ABB RAPID module: lab01_main.mod

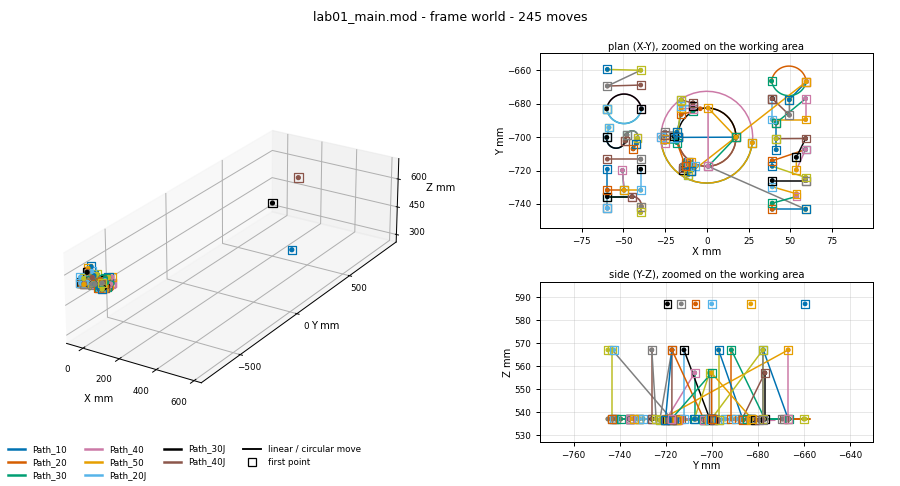
[picture p0: tool path of lab01_main.mod in frame world, 245 of 245 moves have a stored position in this frame; points joined in program order, loops and branches not executed]
MODULE Module1
    CONST robtarget Target_20J:=[[134.579,32.471,0],[1,0,0,0],[0,0,0,0],[9E+09,9E+09,9E+09,9E+09,9E+09,9E+09]];
    CONST robtarget Target_30J:=[[134.579,39.359,0],[1,0,0,0],[0,0,0,0],[9E+09,9E+09,9E+09,9E+09,9E+09,9E+09]];
    CONST robtarget Target_40J:=[[134.579,39.359,0],[1,0,0,0],[0,0,0,0],[9E+09,9E+09,9E+09,9E+09,9E+09,9E+09]];
    CONST robtarget Target_50J:=[[119.781,39.359,0],[1,0,0,0],[0,0,0,0],[9E+09,9E+09,9E+09,9E+09,9E+09,9E+09]];
    CONST robtarget Target_10H:=[[-531.42717004,745,-69.059806194],[0.965925826,0,-0.258819045,0],[0,0,0,0],[9E+09,9E+09,9E+09,9E+09,9E+09,9E+09]];
    CONST robtarget Target_60J:=[[115.729,37.754,0],[1,0,0,0],[0,0,0,0],[9E+09,9E+09,9E+09,9E+09,9E+09,9E+09]];
    CONST robtarget Target_70J:=[[114.303,33.443,0],[1,0,0,0],[0,0,0,0],[9E+09,9E+09,9E+09,9E+09,9E+09,9E+09]];
    CONST robtarget Target_80J:=[[114.692,29.91,0],[1,0,0,0],[0,0,0,0],[9E+09,9E+09,9E+09,9E+09,9E+09,9E+09]];
    CONST robtarget Target_10:=[[606.42717004,0,579.059806194],[0.258819045,0,0.965925826,0],[0,0,0,0],[9E+09,9E+09,9E+09,9E+09,9E+09,9E+09]];
    CONST robtarget Target_30:=[[134.579,39.359,0],[0.707106781,0,0,0.707106781],[0,0,0,0],[9E+09,9E+09,9E+09,9E+09,9E+09,9E+09]];
    CONST robtarget Target_20:=[[134.579,32.471,0],[0.707106781,0,0,0.707106781],[0,0,0,0],[9E+09,9E+09,9E+09,9E+09,9E+09,9E+09]];
    CONST robtarget Target_40:=[[119.781,39.359,0],[0.707106781,0,0,0.707106781],[0,0,0,0],[9E+09,9E+09,9E+09,9E+09,9E+09,9E+09]];
    CONST robtarget Target_50:=[[115.729,37.754,0],[0.707106781,0,0,0.707106781],[0,0,0,0],[9E+09,9E+09,9E+09,9E+09,9E+09,9E+09]];
    CONST robtarget Target_60:=[[114.303,33.443,0],[0.707106781,0,0,0.707106781],[0,0,0,0],[9E+09,9E+09,9E+09,9E+09,9E+09,9E+09]];
    CONST robtarget Target_70:=[[114.692,29.91,0],[0.707106781,0,0,0.707106781],[0,0,0,0],[9E+09,9E+09,9E+09,9E+09,9E+09,9E+09]];
    CONST robtarget Target_80:=[[114.692,29.91,-30],[0.707106781,0,0,0.707106781],[0,0,0,0],[9E+09,9E+09,9E+09,9E+09,9E+09,9E+09]];
    CONST robtarget Target_90:=[[134.579,55.793,0],[0.707106781,0,0,0.707106781],[0,0,0,0],[9E+09,9E+09,9E+09,9E+09,9E+09,9E+09]];
    CONST robtarget Target_100:=[[134.579,43.281,0],[0.707106781,0,0,0.707106781],[0,0,0,0],[9E+09,9E+09,9E+09,9E+09,9E+09,9E+09]];
    CONST robtarget Target_110:=[[124.579,43.281,0],[0.707106781,0,0,0.707106781],[0,0,0,0],[9E+09,9E+09,9E+09,9E+09,9E+09,9E+09]];
    CONST robtarget Target_120:=[[125.551,55.129,0],[0.707106781,0,0,0.707106781],[0,0,0,0],[9E+09,9E+09,9E+09,9E+09,9E+09,9E+09]];
    CONST robtarget Target_130:=[[114.579,43.281,0],[0.707106781,0,0,0.707106781],[0,0,0,0],[9E+09,9E+09,9E+09,9E+09,9E+09,9E+09]];
    CONST robtarget Target_140:=[[114.579,55.793,0],[0.707106781,0,0,0.707106781],[0,0,0,0],[9E+09,9E+09,9E+09,9E+09,9E+09,9E+09]];
    CONST robtarget Target_160:=[[114.579,55.793,-50],[0.707106781,0,0,0.707106781],[0,0,0,0],[9E+09,9E+09,9E+09,9E+09,9E+09,9E+09]];
    CONST robtarget Target_170:=[[134.579,61.806,0],[0.707106781,0,0,0.707106781],[0,0,0,0],[9E+09,9E+09,9E+09,9E+09,9E+09,9E+09]];
    CONST robtarget Target_180:=[[114.579,61.806,0],[0.707106781,0,0,0.707106781],[0,0,0,0],[9E+09,9E+09,9E+09,9E+09,9E+09,9E+09]];
    CONST robtarget Target_190:=[[114.579,61.806,-50],[0.707106781,0,0,0.707106781],[0,0,0,0],[9E+09,9E+09,9E+09,9E+09,9E+09,9E+09]];
    CONST robtarget Target_200:=[[133.639,80.801,0],[0.707106781,0,0,0.707106781],[0,0,0,0],[9E+09,9E+09,9E+09,9E+09,9E+09,9E+09]];
    CONST robtarget Target_210:=[[134.935,74.853,0],[0.707106781,0,0,0.707106781],[0,0,0,0],[9E+09,9E+09,9E+09,9E+09,9E+09,9E+09]];
    CONST robtarget Target_220:=[[133.29,70.023,0],[0.707106781,0,0,0.707106781],[0,0,0,0],[9E+09,9E+09,9E+09,9E+09,9E+09,9E+09]];
    CONST robtarget Target_230:=[[123.833,72.73,0],[0.707106781,0,0,0.707106781],[0,0,0,0],[9E+09,9E+09,9E+09,9E+09,9E+09,9E+09]];
    CONST robtarget Target_240:=[[122.925,76.344,0],[0.707106781,0,0,0.707106781],[0,0,0,0],[9E+09,9E+09,9E+09,9E+09,9E+09,9E+09]];
    CONST robtarget Target_250:=[[119.862,78.808,0],[0.707106781,0,0,0.707106781],[0,0,0,0],[9E+09,9E+09,9E+09,9E+09,9E+09,9E+09]];
    CONST robtarget Target_260:=[[116.524,74.351,0],[0.707106781,0,0,0.707106781],[0,0,0,0],[9E+09,9E+09,9E+09,9E+09,9E+09,9E+09]];
    CONST robtarget Target_270:=[[117.204,71.15,0],[0.707106781,0,0,0.707106781],[0,0,0,0],[9E+09,9E+09,9E+09,9E+09,9E+09,9E+09]];
    CONST robtarget Target_280:=[[119.117,68.078,0],[0.707106781,0,0,0.707106781],[0,0,0,0],[9E+09,9E+09,9E+09,9E+09,9E+09,9E+09]];
    CONST robtarget Target_290:=[[119.117,67.981,-50],[0.707106781,0,0,0.707106781],[0,0,0,0],[9E+09,9E+09,9E+09,9E+09,9E+09,9E+09]];
    CONST robtarget Target_300:=[[135,91.984,0],[0.707106781,0,0,0.707106781],[0,0,0,0],[9E+09,9E+09,9E+09,9E+09,9E+09,9E+09]];
    CONST robtarget Target_310:=[[124.579,83.151,0],[0.707106781,0,0,0.707106781],[0,0,0,0],[9E+09,9E+09,9E+09,9E+09,9E+09,9E+09]];
    CONST robtarget Target_320:=[[114.157,91.984,0],[0.707106781,0,0,0.707106781],[0,0,0,0],[9E+09,9E+09,9E+09,9E+09,9E+09,9E+09]];
    CONST robtarget Target_330:=[[124.579,100.834,0],[0.707106781,0,0,0.707106781],[0,0,0,0],[9E+09,9E+09,9E+09,9E+09,9E+09,9E+09]];
    CONST robtarget Target_340:=[[135,91.984,-50],[0.707106781,0,0,0.707106781],[0,0,0,0],[9E+09,9E+09,9E+09,9E+09,9E+09,9E+09]];
    CONST robtarget Target_360:=[[114.579,106.231,0],[0.707106781,0,0,0.707106781],[0,0,0,0],[9E+09,9E+09,9E+09,9E+09,9E+09,9E+09]];
    CONST robtarget Target_350:=[[134.579,105.639,0],[0.707106781,0,0,0.707106781],[0,0,0,0],[9E+09,9E+09,9E+09,9E+09,9E+09,9E+09]];
    CONST robtarget Target_370:=[[114.579,115.08,0],[0.707106781,0,0,0.707106781],[0,0,0,0],[9E+09,9E+09,9E+09,9E+09,9E+09,9E+09]];
    CONST robtarget Target_380:=[[134.579,115.582,0],[0.707106781,0,0,0.707106781],[0,0,0,0],[9E+09,9E+09,9E+09,9E+09,9E+09,9E+09]];
    CONST robtarget Target_390:=[[134.579,115.582,-50],[0.707106781,0,0,0.707106781],[0,0,0,0],[9E+09,9E+09,9E+09,9E+09,9E+09,9E+09]];
    CONST robtarget Target_400:=[[102.5,75,0],[0.707106781,0,0,0.707106781],[0,0,0,0],[9E+09,9E+09,9E+09,9E+09,9E+09,9E+09]];
    CONST robtarget Target_410:=[[77.953,102.341,0.5],[0.707106781,0,0,0.707106781],[0,0,0,0],[9E+09,9E+09,9E+09,9E+09,9E+09,9E+09]];
    CONST robtarget Target_420:=[[47.704,71.659,0.5],[0.707106781,0,0,0.707106781],[0,0,0,0],[9E+09,9E+09,9E+09,9E+09,9E+09,9E+09]];
    CONST robtarget Target_430:=[[73.18,47.56,0],[0.707106781,0,0,0.707106781],[0,0,0,0],[9E+09,9E+09,9E+09,9E+09,9E+09,9E+09]];
    CONST robtarget Target_440:=[[92.5,75,0],[0.707106781,0,0,0.707106781],[0,0,0,0],[9E+09,9E+09,9E+09,9E+09,9E+09,9E+09]];
    CONST robtarget Target_450:=[[57.5,75,0],[0.707106781,0,0,0.707106781],[0,0,0,0],[9E+09,9E+09,9E+09,9E+09,9E+09,9E+09]];
    CONST robtarget Target_460:=[[78.949,92.049,0],[0.707106781,0,0,0.707106781],[0,0,0,0],[9E+09,9E+09,9E+09,9E+09,9E+09,9E+09]];
    CONST robtarget Target_480:=[[102.5,75,-50],[0.707106781,0,0,0.707106781],[0,0,0,0],[9E+09,9E+09,9E+09,9E+09,9E+09,9E+09]];
    CONST robtarget Target_490:=[[74.168,57.52,0],[0.707106781,0,0,0.707106781],[0,0,0,0],[9E+09,9E+09,9E+09,9E+09,9E+09,9E+09]];
    CONST robtarget Target_500:=[[15.79,31.822,-30],[0.707106781,0,0,0.707106781],[0,0,0,0],[9E+09,9E+09,9E+09,9E+09,9E+09,9E+09]];
    CONST robtarget Target_510:=[[15.79,31.822,0],[0.707106781,0,0,0.707106781],[0,0,0,0],[9E+09,9E+09,9E+09,9E+09,9E+09,9E+09]];
    CONST robtarget Target_520:=[[35.79,31.822,0],[0.707106781,0,0,0.707106781],[0,0,0,0],[9E+09,9E+09,9E+09,9E+09,9E+09,9E+09]];
    CONST robtarget Target_530:=[[35.79,35.453,0],[0.707106781,0,0,0.707106781],[0,0,0,0],[9E+09,9E+09,9E+09,9E+09,9E+09,9E+09]];
    CONST robtarget Target_540:=[[21.301,39.472,0],[0.707106781,0,0,0.707106781],[0,0,0,0],[9E+09,9E+09,9E+09,9E+09,9E+09,9E+09]];
    CONST robtarget Target_550:=[[21.301,41.093,0],[0.707106781,0,0,0.707106781],[0,0,0,0],[9E+09,9E+09,9E+09,9E+09,9E+09,9E+09]];
    CONST robtarget Target_560:=[[35.79,45.274,0],[0.707106781,0,0,0.707106781],[0,0,0,0],[9E+09,9E+09,9E+09,9E+09,9E+09,9E+09]];
    CONST robtarget Target_570:=[[35.79,48.97,0],[0.707106781,0,0,0.707106781],[0,0,0,0],[9E+09,9E+09,9E+09,9E+09,9E+09,9E+09]];
    CONST robtarget Target_580:=[[15.79,48.97,0],[0.707106781,0,0,0.707106781],[0,0,0,0],[9E+09,9E+09,9E+09,9E+09,9E+09,9E+09]];
    CONST robtarget Target_590:=[[15.79,48.97,-30],[0.707106781,0,0,0.707106781],[0,0,0,0],[9E+09,9E+09,9E+09,9E+09,9E+09,9E+09]];
    CONST robtarget Target_600:=[[15.79,50.866,0],[0.707106781,0,0,0.707106781],[0,0,0,0],[9E+09,9E+09,9E+09,9E+09,9E+09,9E+09]];
    CONST robtarget Target_610:=[[35.79,57.608,0],[0.707106781,0,0,0.707106781],[0,0,0,0],[9E+09,9E+09,9E+09,9E+09,9E+09,9E+09]];
    CONST robtarget Target_620:=[[35.79,60.882,0],[0.707106781,0,0,0.707106781],[0,0,0,0],[9E+09,9E+09,9E+09,9E+09,9E+09,9E+09]];
    CONST robtarget Target_630:=[[15.79,67.625,0],[0.707106781,0,0,0.707106781],[0,0,0,0],[9E+09,9E+09,9E+09,9E+09,9E+09,9E+09]];
    CONST robtarget Target_640:=[[15.79,67.625,-20],[0.707106781,0,0,0.707106781],[0,0,0,0],[9E+09,9E+09,9E+09,9E+09,9E+09,9E+09]];
    CONST robtarget Target_650:=[[21.361,55.365,0],[0.707106781,0,0,0.707106781],[0,0,0,0],[9E+09,9E+09,9E+09,9E+09,9E+09,9E+09]];
    CONST robtarget Target_660:=[[21.382,62.997,0],[0.707106781,0,0,0.707106781],[0,0,0,0],[9E+09,9E+09,9E+09,9E+09,9E+09,9E+09]];
    CONST robtarget Target_670:=[[21.382,62.943,-30],[0.707106781,0,0,0.707106781],[0,0,0,0],[9E+09,9E+09,9E+09,9E+09,9E+09,9E+09]];
    CONST robtarget Target_680:=[[15.79,74.189,0],[0.707106781,0,0,0.707106781],[0,0,0,0],[9E+09,9E+09,9E+09,9E+09,9E+09,9E+09]];
    CONST robtarget Target_690:=[[33.424,74.097,0],[0.707106781,0,0,0.707106781],[0,0,0,0],[9E+09,9E+09,9E+09,9E+09,9E+09,9E+09]];
    CONST robtarget Target_700:=[[33.424,74.055,-20],[0.707106781,0,0,0.707106781],[0,0,0,0],[9E+09,9E+09,9E+09,9E+09,9E+09,9E+09]];
    CONST robtarget Target_710:=[[33.424,67.479,0],[0.707106781,0,0,0.707106781],[0,0,0,0],[9E+09,9E+09,9E+09,9E+09,9E+09,9E+09]];
    CONST robtarget Target_720:=[[33.424,83.556,0],[0.707106781,0,0,0.707106781],[0,0,0,0],[9E+09,9E+09,9E+09,9E+09,9E+09,9E+09]];
    CONST robtarget Target_730:=[[33.424,83.556,-30],[0.707106781,0,0,0.707106781],[0,0,0,0],[9E+09,9E+09,9E+09,9E+09,9E+09,9E+09]];
    CONST robtarget Target_740:=[[15.79,98.095,0],[0.707106781,0,0,0.707106781],[0,0,0,0],[9E+09,9E+09,9E+09,9E+09,9E+09,9E+09]];
    CONST robtarget Target_750:=[[15.79,85.582,0],[0.707106781,0,0,0.707106781],[0,0,0,0],[9E+09,9E+09,9E+09,9E+09,9E+09,9E+09]];
    CONST robtarget Target_760:=[[35.79,85.582,0],[0.707106781,0,0,0.707106781],[0,0,0,0],[9E+09,9E+09,9E+09,9E+09,9E+09,9E+09]];
    CONST robtarget Target_770:=[[35.79,98.095,0],[0.707106781,0,0,0.707106781],[0,0,0,0],[9E+09,9E+09,9E+09,9E+09,9E+09,9E+09]];
    CONST robtarget Target_780:=[[35.79,98.095,-20],[0.707106781,0,0,0.707106781],[0,0,0,0],[9E+09,9E+09,9E+09,9E+09,9E+09,9E+09]];
    CONST robtarget Target_790:=[[25.531,88.24,0],[0.707106781,0,0,0.707106781],[0,0,0,0],[9E+09,9E+09,9E+09,9E+09,9E+09,9E+09]];
    CONST robtarget Target_800:=[[25.579,97.43,0],[0.707106781,0,0,0.707106781],[0,0,0,0],[9E+09,9E+09,9E+09,9E+09,9E+09,9E+09]];
    CONST robtarget Target_810:=[[25.579,97.43,-30],[0.707106781,0,0,0.707106781],[0,0,0,0],[9E+09,9E+09,9E+09,9E+09,9E+09,9E+09]];
    CONST robtarget Target_820:=[[15.378,108.24,0],[0.707106781,0,0,0.707106781],[0,0,0,0],[9E+09,9E+09,9E+09,9E+09,9E+09,9E+09]];
    CONST robtarget Target_830:=[[24.545794471,117.51743745,0],[0.707106781,0,0,0.707106781],[0,0,0,0],[9E+09,9E+09,9E+09,9E+09,9E+09,9E+09]];
    CONST robtarget Target_840:=[[36.211188313,108.651374241,0],[0.707106781,0,0,0.707106781],[0,0,0,0],[9E+09,9E+09,9E+09,9E+09,9E+09,9E+09]];
    CONST robtarget Target_850:=[[25.417582154,99.88143745,0],[0.707106781,0,0,0.707106781],[0,0,0,0],[9E+09,9E+09,9E+09,9E+09,9E+09,9E+09]];
    CONST robtarget Target_860:=[[15.378,108.24,-30],[0.707106781,0,0,0.707106781],[0,0,0,0],[9E+09,9E+09,9E+09,9E+09,9E+09,9E+09]];
    CONST robtarget Target_870:=[[86.451,52.441,0.5],[0.707106781,0,0,0.707106781],[0,0,0,0],[9E+09,9E+09,9E+09,9E+09,9E+09,9E+09]];
    CONST robtarget Target_890:=[[89.117,56.754,0.5],[0.707106781,0,0,0.707106781],[0,0,0,0],[9E+09,9E+09,9E+09,9E+09,9E+09,9E+09]];
    CONST robtarget Target_880:=[[89.302,55.354,0.5],[0.707106781,0,0,0.707106781],[0,0,0,0],[9E+09,9E+09,9E+09,9E+09,9E+09,9E+09]];
    CONST robtarget Target_900:=[[88.422,57.436,0.5],[0.707106781,0,0,0.707106781],[0,0,0,0],[9E+09,9E+09,9E+09,9E+09,9E+09,9E+09]];
    CONST robtarget Target_910:=[[87.783,57.66,0.546],[0.707106781,0,0,0.707106781],[0,0,0,0],[9E+09,9E+09,9E+09,9E+09,9E+09,9E+09]];
    CONST robtarget Target_920:=[[87.728,58.612,0.5],[0.707106781,0,0,0.707106781],[0,0,0,0],[9E+09,9E+09,9E+09,9E+09,9E+09,9E+09]];
    CONST robtarget Target_930:=[[87.299,59.362,0.5],[0.707106781,0,0,0.707106781],[0,0,0,0],[9E+09,9E+09,9E+09,9E+09,9E+09,9E+09]];
    CONST robtarget Target_940:=[[86.474,59.997,0.5],[0.707106781,0,0,0.707106781],[0,0,0,0],[9E+09,9E+09,9E+09,9E+09,9E+09,9E+09]];
    CONST robtarget Target_950:=[[85.487,60.183,0.5],[0.707106781,0,0,0.707106781],[0,0,0,0],[9E+09,9E+09,9E+09,9E+09,9E+09,9E+09]];
    CONST robtarget Target_960:=[[84.601,59.985,0.5],[0.707106781,0,0,0.707106781],[0,0,0,0],[9E+09,9E+09,9E+09,9E+09,9E+09,9E+09]];
    CONST robtarget Target_970:=[[81.843,57.842,0.5],[0.707106781,0,0,0.707106781],[0,0,0,0],[9E+09,9E+09,9E+09,9E+09,9E+09,9E+09]];
    CONST robtarget Target_980:=[[84.366,54.885,0.5],[0.707106781,0,0,0.707106781],[0,0,0,0],[9E+09,9E+09,9E+09,9E+09,9E+09,9E+09]];
    CONST robtarget Target_990:=[[87.79,57.696,0.5],[0.707106781,0,0,0.707106781],[0,0,0,0],[9E+09,9E+09,9E+09,9E+09,9E+09,9E+09]];
    CONST robtarget Target_1020:=[[87.797,57.739,-30],[0.707106781,0,0,0.707106781],[0,0,0,0],[9E+09,9E+09,9E+09,9E+09,9E+09,9E+09]];
    CONST robtarget Target_1010:=[[86.451,52.441,0.5],[0.707106781,0,0,0.707106781],[0,0,0,0],[9E+09,9E+09,9E+09,9E+09,9E+09,9E+09]];
    CONST robtarget Target_1030:=[[92.924,71.772,0.5],[0.707106781,0,0,0.707106781],[0,0,0,0],[9E+09,9E+09,9E+09,9E+09,9E+09,9E+09]];
    CONST robtarget Target_1040:=[[100.024,71.772,0.5],[0.707106781,0,0,0.707106781],[0,0,0,0],[9E+09,9E+09,9E+09,9E+09,9E+09,9E+09]];
    CONST robtarget Target_1050:=[[100.024,73.703,0.5],[0.707106781,0,0,0.707106781],[0,0,0,0],[9E+09,9E+09,9E+09,9E+09,9E+09,9E+09]];
    CONST robtarget Target_1060:=[[94.605,74.279,0.5],[0.707106781,0,0,0.707106781],[0,0,0,0],[9E+09,9E+09,9E+09,9E+09,9E+09,9E+09]];
    CONST robtarget Target_1070:=[[94.605,75.424,0.5],[0.707106781,0,0,0.707106781],[0,0,0,0],[9E+09,9E+09,9E+09,9E+09,9E+09,9E+09]];
    CONST robtarget Target_1080:=[[100.024,76.047,0.5],[0.707106781,0,0,0.707106781],[0,0,0,0],[9E+09,9E+09,9E+09,9E+09,9E+09,9E+09]];
    CONST robtarget Target_1090:=[[100.024,78.002,0.5],[0.707106781,0,0,0.707106781],[0,0,0,0],[9E+09,9E+09,9E+09,9E+09,9E+09,9E+09]];
    CONST robtarget Target_1100:=[[92.924,78.002,0.5],[0.707106781,0,0,0.707106781],[0,0,0,0],[9E+09,9E+09,9E+09,9E+09,9E+09,9E+09]];
    CONST robtarget Target_1110:=[[92.924,78.002,-30],[0.707106781,0,0,0.707106781],[0,0,0,0],[9E+09,9E+09,9E+09,9E+09,9E+09,9E+09]];
    CONST robtarget Target_1120:=[[90.373,88.629,0.5],[0.707106781,0,0,0.707106781],[0,0,0,0],[9E+09,9E+09,9E+09,9E+09,9E+09,9E+09]];
    CONST robtarget Target_1130:=[[83.273,90.441,0],[0.707106781,0,0,0.707106781],[0,0,0,0],[9E+09,9E+09,9E+09,9E+09,9E+09,9E+09]];
    CONST robtarget Target_1140:=[[83.273,92.124,0.5],[0.707106781,0,0,0.707106781],[0,0,0,0],[9E+09,9E+09,9E+09,9E+09,9E+09,9E+09]];
    CONST robtarget Target_1150:=[[90.373,92.156,0.5],[0.707106781,0,0,0.707106781],[0,0,0,0],[9E+09,9E+09,9E+09,9E+09,9E+09,9E+09]];
    CONST robtarget Target_1160:=[[90.373,93.77,0.5],[0.707106781,0,0,0.707106781],[0,0,0,0],[9E+09,9E+09,9E+09,9E+09,9E+09,9E+09]];
    CONST robtarget Target_1170:=[[83.273,93.784,0.5],[0.707106781,0,0,0.707106781],[0,0,0,0],[9E+09,9E+09,9E+09,9E+09,9E+09,9E+09]];
    CONST robtarget Target_1180:=[[83.273,95.476,0.5],[0.707106781,0,0,0.707106781],[0,0,0,0],[9E+09,9E+09,9E+09,9E+09,9E+09,9E+09]];
    CONST robtarget Target_1190:=[[90.367,97.258,0.5],[0.707106781,0,0,0.707106781],[0,0,0,0],[9E+09,9E+09,9E+09,9E+09,9E+09,9E+09]];
    CONST robtarget Target_1200:=[[90.307,97.243,-30],[0.707106781,0,0,0.707106781],[0,0,0,0],[9E+09,9E+09,9E+09,9E+09,9E+09,9E+09]];
    CONST robtarget Target_1210:=[[92.5,74.875,0],[0.707106781,0,0,0.707106781],[0,0,0,0],[9E+09,9E+09,9E+09,9E+09,9E+09,9E+09]];
    CONST robtarget Target_1220:=[[57.5,75.002,0],[0.707106781,0,0,0.707106781],[0,0,0,0],[9E+09,9E+09,9E+09,9E+09,9E+09,9E+09]];
    CONST robtarget Target_1230:=[[57.5,74.962,-20],[0.707106781,0,0,0.707106781],[0,0,0,0],[9E+09,9E+09,9E+09,9E+09,9E+09,9E+09]];
    CONST robtarget Target_1240:=[[74.192,57.519,0],[0.707106781,0,0,0.707106781],[0,0,0,0],[9E+09,9E+09,9E+09,9E+09,9E+09,9E+09]];
    CONST robtarget Target_1250:=[[74.241,92.484,0],[0.707106781,0,0,0.707106781],[0,0,0,0],[9E+09,9E+09,9E+09,9E+09,9E+09,9E+09]];
    PERS tooldata Tool_JM:=[TRUE,[[36.916,0,136.94],[0.965925826,0,0.258819045,0]],[0.1,[0,0,1],[1,0,0,0],0,0,0]];
    TASK PERS wobjdata Workobject_4:=[FALSE,TRUE,"",[[0,-100,27],[1,0,0,0]],[[75,-675,510],[0,0,1,0]]];
    CONST robtarget Target_1260:=[[134.579,32.471,-30],[0.707106781,0,0,0.707106781],[0,0,0,0],[9E+09,9E+09,9E+09,9E+09,9E+09,9E+09]];
    CONST robtarget Target_1270:=[[74.522025646,1604.781854023,155.867635961],[0.664355676,-0.23027169,-0.237213164,-0.670325592],[1,0,-1,0],[9E+09,9E+09,9E+09,9E+09,9E+09,9E+09]];
    CONST robtarget Target_1280:=[[-35.006958294,1674.86910456,16.96090151],[0.661721738,-0.310193659,-0.350423362,-0.585753961],[0,0,-1,1],[9E+09,9E+09,9E+09,9E+09,9E+09,9E+09]];

    PROC main()

        WHILE TRUE DO

            IF DI_01 = 1 THEN
                Set DO_01;
                WaitTime(4.9);
                Reset DO_01;
                Path_10;
                Path_1110;
                Path_20J;
                Path_30J;
                Path_40J;
                Path_50J;
                Path_60;
                Path_70E;
                Path_80E;
                Path_90E;
                Path_100E;
                Path_110E;
                Path_120E;
                Path_120;
                Path_130I;
                Path_140;
                Path_150S;
                Path_160S;
                Path_170S;
                Path_180S;
                Path_190S;
                Path_200S;
                Path_210;
                Path_220O;
                Path_230O;
                Path_240;
                Path_250N;
                Path_260N;
                Path_270N;
                Path_280;
                Path_290L;
                Path_300;
                Path_310;
                Path_320;
                Path_330;
                Path_340;
                Path_350;
                Path_360;
                Path_370;
                Path_380;
                Path_390;
                Path_400;
                Path_410;
                Path_420;
                Path_430;
                Path_440;
                Path_450;
                Path_460;
                Path_470;
                Path_480;
                Path_490;
                Path_500;
                Path_510;
                Path_520;
                Path_530;
                Path_540;
                Path_550;
                Path_560;
                Path_570;
                Path_580;
                Path_590;
                Path_600;
                Path_610;
                Path_620;
                Path_630;
                Path_640;
                Path_650;
                Path_660;
                Path_670;
                Path_680;
                Path_690;
                Path_700;
                Path_710;
                Path_720;
                Path_730;
                Path_740;
                Path_750;
                Path_760;
                Path_770;
                Path_780;
                Path_790;
                Path_800;
                Path_810;
                Path_820;
                Path_830;
                Path_840;
                Path_850;
                Path_860;
                Path_870;
                Path_880;
                Path_890;
                Path_900;
                Path_910;
                Path_920;
                Path_930;
                Path_940;
                Path_950;
                Path_960;
                Path_970;
                Path_980;
                Path_990;
                Path_1000;
                Path_1010;
                Path_1020;
                Path_1030;
                Path_1040;
                Path_1050;
                Path_1060;
                Path_1070;
                Path_1080;
                Path_1090;
                Path_1100;


                Path_10;

                Reset DO_01;


            ENDIF

            IF DI_02 = 1 THEN
                Set DO_02;
                Path_1130;
                Reset DO_02;

            ENDIF




        ENDWHILE

    ENDPROC
    PROC Path_10()
        MoveJ Target_10,v100,z10,Tool_JM\WObj:=wobj0;
    ENDPROC
    PROC Path_20()
        MoveL Target_20,v100,z10,Tool_JM\WObj:=Workobject_4;
        MoveL Target_30,v100,z10,Tool_JM\WObj:=Workobject_4;
    ENDPROC
    PROC Path_30()
        MoveL Target_30,v100,z10,Tool_JM\WObj:=Workobject_4;
        MoveL Target_40,v100,z10,Tool_JM\WObj:=Workobject_4;
    ENDPROC
    PROC Path_40()
        MoveJ Target_40,v100,z10,Tool_JM\WObj:=Workobject_4;
        MoveC Target_50,Target_60,v100,z10,Tool_JM\WObj:=Workobject_4;
    ENDPROC
    PROC Path_50()
        MoveL Target_60,v100,z10,Tool_JM\WObj:=Workobject_4;
        MoveL Target_70,v100,z10,Tool_JM\WObj:=Workobject_4;
    ENDPROC
    PROC Path_20J()
        MoveL Target_20,v100,z10,Tool_JM\WObj:=Workobject_4;
        MoveL Target_30,v100,z10,Tool_JM\WObj:=Workobject_4;
    ENDPROC
    PROC Path_30J()
        MoveL Target_30,v100,z10,Tool_JM\WObj:=Workobject_4;
        MoveL Target_40,v100,z10,Tool_JM\WObj:=Workobject_4;
    ENDPROC
    PROC Path_40J()
        MoveJ Target_40,v100,z10,Tool_JM\WObj:=Workobject_4;
        MoveC Target_50,Target_60,v100,z10,Tool_JM\WObj:=Workobject_4;
    ENDPROC
    PROC Path_50J()
        MoveL Target_60,v100,z10,Tool_JM\WObj:=Workobject_4;
        MoveL Target_70,v100,z10,Tool_JM\WObj:=Workobject_4;
    ENDPROC
    PROC Path_60()
        MoveL Target_80,v100,z10,Tool_JM\WObj:=Workobject_4;
    ENDPROC
    PROC Path_70E()
        MoveL Target_90,v100,z10,Tool_JM\WObj:=Workobject_4;
        MoveL Target_100,v100,z10,Tool_JM\WObj:=Workobject_4;
    ENDPROC
    PROC Path_80E()
        MoveL Target_100,v100,z10,Tool_JM\WObj:=Workobject_4;
        MoveL Target_110,v100,z10,Tool_JM\WObj:=Workobject_4;
    ENDPROC
    PROC Path_90E()
        MoveL Target_110,v100,z10,Tool_JM\WObj:=Workobject_4;
        MoveL Target_120,v100,z10,Tool_JM\WObj:=Workobject_4;
    ENDPROC
    PROC Path_100E()
        MoveL Target_120,v100,z10,Tool_JM\WObj:=Workobject_4;
        MoveL Target_110,v100,z10,Tool_JM\WObj:=Workobject_4;
    ENDPROC
    PROC Path_110E()
        MoveL Target_110,v100,z10,Tool_JM\WObj:=Workobject_4;
        MoveL Target_130,v100,z10,Tool_JM\WObj:=Workobject_4;
    ENDPROC
    PROC Path_120E()
        MoveL Target_130,v100,z10,Tool_JM\WObj:=Workobject_4;
        MoveL Target_140,v100,z10,Tool_JM\WObj:=Workobject_4;
    ENDPROC
    PROC Path_120()
        MoveJ Target_160,v100,z10,Tool_JM\WObj:=Workobject_4;
    ENDPROC
    PROC Path_130I()
        MoveL Target_170,v100,z10,Tool_JM\WObj:=Workobject_4;
        MoveL Target_180,v100,z10,Tool_JM\WObj:=Workobject_4;
    ENDPROC
    PROC Path_140()
        MoveJ Target_190,v100,z10,Tool_JM\WObj:=Workobject_4;
    ENDPROC
    PROC Path_150()
        MoveL Target_200,v100,z10,Tool_JM\WObj:=Workobject_4;
        MoveL Target_210,v100,z10,Tool_JM\WObj:=Workobject_4;
    ENDPROC
    PROC Path_160()
        MoveJ Target_210,v100,z10,Tool_JM\WObj:=Workobject_4;
        MoveC Target_220,Target_230,v100,z10,Tool_JM\WObj:=Workobject_4;
    ENDPROC
    PROC Path_170()
        MoveL Target_230,v100,z10,Tool_JM\WObj:=Workobject_4;
        MoveL Target_240,v100,z10,Tool_JM\WObj:=Workobject_4;
    ENDPROC
    PROC Path_180()
        MoveJ Target_240,v100,z10,Tool_JM\WObj:=Workobject_4;
        MoveC Target_250,Target_260,v100,z10,Tool_JM\WObj:=Workobject_4;
    ENDPROC
    PROC Path_190()
        MoveL Target_260,v100,z10,Tool_JM\WObj:=Workobject_4;
        MoveL Target_270,v100,z10,Tool_JM\WObj:=Workobject_4;
    ENDPROC
    PROC Path_200()
        MoveL Target_270,v100,z10,Tool_JM\WObj:=Workobject_4;
        MoveL Target_280,v100,z10,Tool_JM\WObj:=Workobject_4;
    ENDPROC
    PROC Path_150S()
        MoveL Target_200,v100,z10,Tool_JM\WObj:=Workobject_4;
        MoveL Target_210,v100,z10,Tool_JM\WObj:=Workobject_4;
    ENDPROC
    PROC Path_160S()
        MoveJ Target_210,v100,z10,Tool_JM\WObj:=Workobject_4;
        MoveC Target_220,Target_230,v100,z10,Tool_JM\WObj:=Workobject_4;
    ENDPROC
    PROC Path_170S()
        MoveL Target_230,v100,z10,Tool_JM\WObj:=Workobject_4;
        MoveL Target_240,v100,z10,Tool_JM\WObj:=Workobject_4;
    ENDPROC
    PROC Path_180S()
        MoveJ Target_240,v100,z10,Tool_JM\WObj:=Workobject_4;
        MoveC Target_250,Target_260,v100,z10,Tool_JM\WObj:=Workobject_4;
    ENDPROC
    PROC Path_190S()
        MoveL Target_260,v100,z10,Tool_JM\WObj:=Workobject_4;
        MoveL Target_270,v100,z10,Tool_JM\WObj:=Workobject_4;
    ENDPROC
    PROC Path_200S()
        MoveL Target_270,v100,z10,Tool_JM\WObj:=Workobject_4;
        MoveL Target_280,v100,z10,Tool_JM\WObj:=Workobject_4;
    ENDPROC
    PROC Path_210()
        MoveL Target_290,v100,z10,Tool_JM\WObj:=Workobject_4;
    ENDPROC
    PROC Path_220()
        MoveJ Target_300,v100,z10,Tool_JM\WObj:=Workobject_4;
        MoveC Target_310,Target_320,v100,z10,Tool_JM\WObj:=Workobject_4;
    ENDPROC
    PROC Path_230()
        MoveJ Target_320,v100,z10,Tool_JM\WObj:=Workobject_4;
        MoveC Target_330,Target_300,v100,z10,Tool_JM\WObj:=Workobject_4;

    ENDPROC
    PROC Path_240()
        MoveJ Target_340,v100,z10,Tool_JM\WObj:=Workobject_4;
    ENDPROC
    PROC Path_220O()
        MoveJ Target_300,v100,z10,Tool_JM\WObj:=Workobject_4;
        MoveC Target_310,Target_320,v100,z10,Tool_JM\WObj:=Workobject_4;
    ENDPROC
    PROC Path_230O()
        MoveJ Target_320,v100,z10,Tool_JM\WObj:=Workobject_4;
        MoveC Target_330,Target_300,v100,z10,Tool_JM\WObj:=Workobject_4;
    ENDPROC
    PROC Path_250N()
        MoveL Target_360,v100,z10,Tool_JM\WObj:=Workobject_4;
        MoveL Target_350,v100,z10,Tool_JM\WObj:=Workobject_4;
    ENDPROC
    PROC Path_260N()
        MoveL Target_350,v100,z10,Tool_JM\WObj:=Workobject_4;
        MoveL Target_370,v100,z10,Tool_JM\WObj:=Workobject_4;
    ENDPROC
    PROC Path_270N()
        MoveL Target_370,v100,z10,Tool_JM\WObj:=Workobject_4;
        MoveL Target_380,v100,z10,Tool_JM\WObj:=Workobject_4;
    ENDPROC
    PROC Path_280()
        MoveL Target_390,v100,z10,Tool_JM\WObj:=Workobject_4;
    ENDPROC
    PROC Path_290()
        MoveJ Target_440,v100,z10,Tool_JM\WObj:=Workobject_4;
        MoveC Target_450,Target_460,v100,z10,Tool_JM\WObj:=Workobject_4;

    ENDPROC
    PROC Path_300()
        MoveJ Target_420,v100,z10,Tool_JM\WObj:=Workobject_4;
        MoveC Target_430,Target_400,v100,z10,Tool_JM\WObj:=Workobject_4;
    ENDPROC
    PROC Path_290L()
        MoveJ Target_400,v100,z10,Tool_JM\WObj:=Workobject_4;
        MoveC Target_410,Target_420,v100,z10,Tool_JM\WObj:=Workobject_4;
    ENDPROC
    PROC Path_300L()
        MoveJ Target_420,v100,z10,Tool_JM\WObj:=Workobject_4;
        MoveC Target_430,Target_400,v100,z10,Tool_JM\WObj:=Workobject_4;
    ENDPROC
    PROC Path_310()
        MoveL Target_480,v100,z10,Tool_JM\WObj:=Workobject_4;
    ENDPROC
    PROC Path_320()
        MoveJ Target_440,v100,z10,Tool_JM\WObj:=Workobject_4;
        MoveC Target_460,Target_450,v100,z10,Tool_JM\WObj:=Workobject_4;

    ENDPROC
    PROC Path_330()
        MoveJ Target_450,v100,z10,Tool_JM\WObj:=Workobject_4;
        MoveC Target_490,Target_440,v100,z10,Tool_JM\WObj:=Workobject_4;

    ENDPROC
    PROC Path_340()
        MoveL Target_490,v100,z10,Tool_JM\WObj:=Workobject_4;
        MoveL Target_500,v100,z10,Tool_JM\WObj:=Workobject_4;
    ENDPROC
    PROC Path_350()
        MoveL Target_500,v100,z10,Tool_JM\WObj:=Workobject_4;
        MoveL Target_510,v100,z10,Tool_JM\WObj:=Workobject_4;
    ENDPROC
    PROC Path_360()
        MoveL Target_510,v100,z10,Tool_JM\WObj:=Workobject_4;
        MoveL Target_520,v100,z10,Tool_JM\WObj:=Workobject_4;
    ENDPROC
    PROC Path_370()
        MoveL Target_520,v100,z10,Tool_JM\WObj:=Workobject_4;
        MoveL Target_530,v100,z10,Tool_JM\WObj:=Workobject_4;
    ENDPROC
    PROC Path_380()
        MoveL Target_530,v100,z10,Tool_JM\WObj:=Workobject_4;
        MoveL Target_540,v100,z10,Tool_JM\WObj:=Workobject_4;
    ENDPROC
    PROC Path_390()
        MoveL Target_540,v100,z10,Tool_JM\WObj:=Workobject_4;
        MoveL Target_550,v100,z10,Tool_JM\WObj:=Workobject_4;
    ENDPROC
    PROC Path_400()
        MoveL Target_550,v100,z10,Tool_JM\WObj:=Workobject_4;
        MoveL Target_560,v100,z10,Tool_JM\WObj:=Workobject_4;
    ENDPROC
    PROC Path_410()
        MoveL Target_560,v100,z10,Tool_JM\WObj:=Workobject_4;
        MoveL Target_570,v100,z10,Tool_JM\WObj:=Workobject_4;
    ENDPROC
    PROC Path_420()
        MoveL Target_570,v100,z10,Tool_JM\WObj:=Workobject_4;
        MoveL Target_580,v100,z10,Tool_JM\WObj:=Workobject_4;
    ENDPROC
    PROC Path_430()
        MoveL Target_580,v100,z10,Tool_JM\WObj:=Workobject_4;
        MoveL Target_590,v100,z10,Tool_JM\WObj:=Workobject_4;
    ENDPROC
    PROC Path_440()
        MoveL Target_590,v100,z10,Tool_JM\WObj:=Workobject_4;
        MoveL Target_600,v100,z10,Tool_JM\WObj:=Workobject_4;
    ENDPROC
    PROC Path_450()
        MoveL Target_600,v100,z10,Tool_JM\WObj:=Workobject_4;
        MoveL Target_610,v100,z10,Tool_JM\WObj:=Workobject_4;
    ENDPROC
    PROC Path_460()
        MoveL Target_610,v100,z10,Tool_JM\WObj:=Workobject_4;
        MoveL Target_620,v100,z10,Tool_JM\WObj:=Workobject_4;
    ENDPROC
    PROC Path_470()
        MoveL Target_620,v100,z10,Tool_JM\WObj:=Workobject_4;
        MoveL Target_630,v100,z10,Tool_JM\WObj:=Workobject_4;
    ENDPROC
    PROC Path_480()
        MoveL Target_630,v100,z10,Tool_JM\WObj:=Workobject_4;
        MoveL Target_640,v100,z10,Tool_JM\WObj:=Workobject_4;
    ENDPROC
    PROC Path_490()
        MoveL Target_640,v100,z10,Tool_JM\WObj:=Workobject_4;
        MoveL Target_650,v100,z10,Tool_JM\WObj:=Workobject_4;
    ENDPROC
    PROC Path_500()
        MoveL Target_650,v100,z10,Tool_JM\WObj:=Workobject_4;
        MoveL Target_660,v100,z10,Tool_JM\WObj:=Workobject_4;
    ENDPROC
    PROC Path_510()
        MoveL Target_660,v100,z10,Tool_JM\WObj:=Workobject_4;
        MoveL Target_670,v100,z10,Tool_JM\WObj:=Workobject_4;
    ENDPROC
    PROC Path_520()
        MoveL Target_670,v100,z10,Tool_JM\WObj:=Workobject_4;
        MoveL Target_680,v100,z10,Tool_JM\WObj:=Workobject_4;
    ENDPROC
    PROC Path_530()
        MoveL Target_680,v100,z10,Tool_JM\WObj:=Workobject_4;
        MoveL Target_690,v100,z10,Tool_JM\WObj:=Workobject_4;
    ENDPROC
    PROC Path_540()
        MoveL Target_690,v100,z10,Tool_JM\WObj:=Workobject_4;
        MoveL Target_700,v100,z10,Tool_JM\WObj:=Workobject_4;
    ENDPROC
    PROC Path_550()
        MoveL Target_700,v100,z10,Tool_JM\WObj:=Workobject_4;
        MoveL Target_710,v100,z10,Tool_JM\WObj:=Workobject_4;
    ENDPROC
    PROC Path_560()
        MoveL Target_710,v100,z10,Tool_JM\WObj:=Workobject_4;
        MoveL Target_720,v100,z10,Tool_JM\WObj:=Workobject_4;
    ENDPROC
    PROC Path_570()
        MoveL Target_720,v100,z10,Tool_JM\WObj:=Workobject_4;
        MoveL Target_730,v100,z10,Tool_JM\WObj:=Workobject_4;
    ENDPROC
    PROC Path_580()
        MoveL Target_730,v100,z10,Tool_JM\WObj:=Workobject_4;
        MoveL Target_740,v100,z10,Tool_JM\WObj:=Workobject_4;
    ENDPROC
    PROC Path_590()
        MoveL Target_740,v100,z10,Tool_JM\WObj:=Workobject_4;
        MoveL Target_750,v100,z10,Tool_JM\WObj:=Workobject_4;
    ENDPROC
    PROC Path_600()
        MoveL Target_750,v100,z10,Tool_JM\WObj:=Workobject_4;
        MoveL Target_760,v100,z10,Tool_JM\WObj:=Workobject_4;
    ENDPROC
    PROC Path_610()
        MoveL Target_760,v100,z10,Tool_JM\WObj:=Workobject_4;
        MoveL Target_770,v100,z10,Tool_JM\WObj:=Workobject_4;
    ENDPROC
    PROC Path_620()
        MoveL Target_770,v100,z10,Tool_JM\WObj:=Workobject_4;
        MoveL Target_780,v100,z10,Tool_JM\WObj:=Workobject_4;
    ENDPROC
    PROC Path_630()
        MoveL Target_780,v100,z10,Tool_JM\WObj:=Workobject_4;
        MoveL Target_790,v100,z10,Tool_JM\WObj:=Workobject_4;
    ENDPROC
    PROC Path_640()
        MoveL Target_790,v100,z10,Tool_JM\WObj:=Workobject_4;
        MoveL Target_800,v100,z10,Tool_JM\WObj:=Workobject_4;
    ENDPROC
    PROC Path_650()
        MoveL Target_800,v100,z10,Tool_JM\WObj:=Workobject_4;
        MoveL Target_810,v100,z10,Tool_JM\WObj:=Workobject_4;
    ENDPROC
    PROC Path_660()
        MoveL Target_810,v100,z10,Tool_JM\WObj:=Workobject_4;
        MoveL Target_820,v100,z10,Tool_JM\WObj:=Workobject_4;
    ENDPROC
    PROC Path_670()
        MoveJ Target_820,v100,z10,Tool_JM\WObj:=Workobject_4;
        MoveC Target_830,Target_840,v100,z10,Tool_JM\WObj:=Workobject_4;
    ENDPROC
    PROC Path_680()
        MoveJ Target_840,v100,z10,Tool_JM\WObj:=Workobject_4;
        MoveC Target_850,Target_820,v100,z10,Tool_JM\WObj:=Workobject_4;
    ENDPROC
    PROC Path_690()
        MoveL Target_820,v100,z10,Tool_JM\WObj:=Workobject_4;
        MoveL Target_860,v100,z10,Tool_JM\WObj:=Workobject_4;
    ENDPROC
    PROC Path_700()
        MoveL Target_860,v100,z10,Tool_JM\WObj:=Workobject_4;
        MoveL Target_870,v100,z10,Tool_JM\WObj:=Workobject_4;
    ENDPROC
    PROC Path_710()
        MoveL Target_870,v100,z10,Tool_JM\WObj:=Workobject_4;
        MoveL Target_880,v100,z10,Tool_JM\WObj:=Workobject_4;
    ENDPROC
    PROC Path_720()
        MoveL Target_880,v100,z10,Tool_JM\WObj:=Workobject_4;
        MoveL Target_890,v100,z10,Tool_JM\WObj:=Workobject_4;
    ENDPROC
    PROC Path_730()
        MoveL Target_890,v100,z10,Tool_JM\WObj:=Workobject_4;
        MoveL Target_900,v100,z10,Tool_JM\WObj:=Workobject_4;
    ENDPROC
    PROC Path_740()
        MoveL Target_900,v100,z10,Tool_JM\WObj:=Workobject_4;
        MoveL Target_910,v100,z10,Tool_JM\WObj:=Workobject_4;
    ENDPROC
    PROC Path_750()
        MoveL Target_910,v100,z10,Tool_JM\WObj:=Workobject_4;
        MoveL Target_920,v100,z10,Tool_JM\WObj:=Workobject_4;
    ENDPROC
    PROC Path_760()
        MoveL Target_920,v100,z10,Tool_JM\WObj:=Workobject_4;
        MoveL Target_930,v100,z10,Tool_JM\WObj:=Workobject_4;
    ENDPROC
    PROC Path_770()
        MoveL Target_930,v100,z10,Tool_JM\WObj:=Workobject_4;
        MoveL Target_940,v100,z10,Tool_JM\WObj:=Workobject_4;
    ENDPROC
    PROC Path_780()
        MoveL Target_940,v100,z10,Tool_JM\WObj:=Workobject_4;
        MoveL Target_950,v100,z10,Tool_JM\WObj:=Workobject_4;
    ENDPROC
    PROC Path_790()
        MoveL Target_950,v100,z10,Tool_JM\WObj:=Workobject_4;
        MoveL Target_960,v100,z10,Tool_JM\WObj:=Workobject_4;
    ENDPROC
    PROC Path_800()
        MoveL Target_960,v100,z10,Tool_JM\WObj:=Workobject_4;
        MoveL Target_970,v100,z10,Tool_JM\WObj:=Workobject_4;
    ENDPROC
    PROC Path_810()
        MoveL Target_970,v100,z10,Tool_JM\WObj:=Workobject_4;
        MoveL Target_980,v100,z10,Tool_JM\WObj:=Workobject_4;
    ENDPROC
    PROC Path_820()
        MoveL Target_980,v100,z10,Tool_JM\WObj:=Workobject_4;
        MoveL Target_990,v100,z10,Tool_JM\WObj:=Workobject_4;
    ENDPROC
    PROC Path_830()
        MoveL Target_990,v100,z10,Tool_JM\WObj:=Workobject_4;
        MoveL Target_1020,v100,z10,Tool_JM\WObj:=Workobject_4;
    ENDPROC
    PROC Path_840()
        MoveL Target_1020,v100,z10,Tool_JM\WObj:=Workobject_4;
        MoveL Target_1010,v100,z10,Tool_JM\WObj:=Workobject_4;
    ENDPROC
    PROC Path_850()
        MoveL Target_1010,v100,z10,Tool_JM\WObj:=Workobject_4;
        MoveL Target_980,v100,z10,Tool_JM\WObj:=Workobject_4;
    ENDPROC
    PROC Path_860()
        MoveL Target_980,v100,z10,Tool_JM\WObj:=Workobject_4;
        MoveL Target_1020,v100,z10,Tool_JM\WObj:=Workobject_4;
    ENDPROC
    PROC Path_870()
        MoveL Target_1020,v100,z10,Tool_JM\WObj:=Workobject_4;
        MoveL Target_1030,v100,z10,Tool_JM\WObj:=Workobject_4;
    ENDPROC
    PROC Path_880()
        MoveL Target_1030,v100,z10,Tool_JM\WObj:=Workobject_4;
        MoveL Target_1040,v100,z10,Tool_JM\WObj:=Workobject_4;
    ENDPROC
    PROC Path_890()
        MoveL Target_1040,v100,z10,Tool_JM\WObj:=Workobject_4;
        MoveL Target_1050,v100,z10,Tool_JM\WObj:=Workobject_4;
    ENDPROC
    PROC Path_900()
        MoveL Target_1050,v100,z10,Tool_JM\WObj:=Workobject_4;
        MoveL Target_1060,v100,z10,Tool_JM\WObj:=Workobject_4;
    ENDPROC
    PROC Path_910()
        MoveL Target_1060,v100,z10,Tool_JM\WObj:=Workobject_4;
        MoveL Target_1070,v100,z10,Tool_JM\WObj:=Workobject_4;
    ENDPROC
    PROC Path_920()
        MoveL Target_1070,v100,z10,Tool_JM\WObj:=Workobject_4;
        MoveL Target_1080,v100,z10,Tool_JM\WObj:=Workobject_4;
    ENDPROC
    PROC Path_930()
        MoveL Target_1080,v100,z10,Tool_JM\WObj:=Workobject_4;
        MoveL Target_1090,v100,z10,Tool_JM\WObj:=Workobject_4;
    ENDPROC
    PROC Path_940()
        MoveL Target_1090,v100,z10,Tool_JM\WObj:=Workobject_4;
        MoveL Target_1100,v100,z10,Tool_JM\WObj:=Workobject_4;
    ENDPROC
    PROC Path_950()
        MoveL Target_1100,v100,z10,Tool_JM\WObj:=Workobject_4;
        MoveL Target_1110,v100,z10,Tool_JM\WObj:=Workobject_4;
    ENDPROC
    PROC Path_960()
        MoveL Target_1110,v100,z10,Tool_JM\WObj:=Workobject_4;
        MoveL Target_1120,v100,z10,Tool_JM\WObj:=Workobject_4;
    ENDPROC
    PROC Path_970()
        MoveL Target_1120,v100,z10,Tool_JM\WObj:=Workobject_4;
        MoveL Target_1130,v100,z10,Tool_JM\WObj:=Workobject_4;
    ENDPROC
    PROC Path_980()
        MoveL Target_1130,v100,z10,Tool_JM\WObj:=Workobject_4;
        MoveL Target_1140,v100,z10,Tool_JM\WObj:=Workobject_4;
    ENDPROC
    PROC Path_990()
        MoveL Target_1140,v100,z10,Tool_JM\WObj:=Workobject_4;
        MoveL Target_1150,v100,z10,Tool_JM\WObj:=Workobject_4;
    ENDPROC
    PROC Path_1000()
        MoveL Target_1150,v100,z10,Tool_JM\WObj:=Workobject_4;
        MoveL Target_1160,v100,z10,Tool_JM\WObj:=Workobject_4;
    ENDPROC
    PROC Path_1010()
        MoveL Target_1160,v100,z10,Tool_JM\WObj:=Workobject_4;
        MoveL Target_1170,v100,z10,Tool_JM\WObj:=Workobject_4;
    ENDPROC
    PROC Path_1020()
        MoveL Target_1170,v100,z10,Tool_JM\WObj:=Workobject_4;
        MoveL Target_1180,v100,z10,Tool_JM\WObj:=Workobject_4;
    ENDPROC
    PROC Path_1030()
        MoveL Target_1180,v100,z10,Tool_JM\WObj:=Workobject_4;
        MoveL Target_1190,v100,z10,Tool_JM\WObj:=Workobject_4;
    ENDPROC
    PROC Path_1040()
        MoveL Target_1190,v100,z10,Tool_JM\WObj:=Workobject_4;
        MoveL Target_1200,v100,z10,Tool_JM\WObj:=Workobject_4;
    ENDPROC
    PROC Path_1050()
        MoveL Target_1200,v100,z10,Tool_JM\WObj:=Workobject_4;
        MoveL Target_1210,v100,z10,Tool_JM\WObj:=Workobject_4;
    ENDPROC
    PROC Path_1060()
        MoveL Target_1210,v100,z10,Tool_JM\WObj:=Workobject_4;
        MoveL Target_1220,v100,z10,Tool_JM\WObj:=Workobject_4;
    ENDPROC
    PROC Path_1070()
        MoveL Target_1220,v100,z10,Tool_JM\WObj:=Workobject_4;
        MoveL Target_1230,v100,z10,Tool_JM\WObj:=Workobject_4;
    ENDPROC
    PROC Path_1080()
        MoveL Target_1230,v100,z10,Tool_JM\WObj:=Workobject_4;
        MoveL Target_1240,v100,z10,Tool_JM\WObj:=Workobject_4;
    ENDPROC
    PROC Path_1090()
        MoveL Target_1240,v100,z10,Tool_JM\WObj:=Workobject_4;
        MoveL Target_1250,v100,z10,Tool_JM\WObj:=Workobject_4;
    ENDPROC
    PROC Path_1100()
        MoveL Target_1250,v100,z10,Tool_JM\WObj:=Workobject_4;
        MoveL Target_1230,v100,z10,Tool_JM\WObj:=Workobject_4;
    ENDPROC
    PROC Path_1110()
        MoveJ Target_1260,v100,z10,Tool_JM\WObj:=Workobject_4;
    ENDPROC
    PROC Path_1120()
        MoveL Target_1270,v1000,z100,Tool_JM\WObj:=Workobject_4;
    ENDPROC
    PROC Path_1130()
        MoveL Target_1280,v100,z10,Tool_JM\WObj:=Workobject_4;
    ENDPROC
ENDMODULE
